TYPE ST_AccessPanel :
STRUCT
	inputs : ST_AccessPanelInputs;
	outputs : ST_AccessPanelOutputs;
END_STRUCT
END_TYPE

(* stored: Version 1.1.0.1, ProductVersion 3.1.4024.4
   DUT ST_AccessPanel: Id {a4a5c948-79a4-4b5c-810d-e6a1bbaeea3e} *)
